PROGRAM POU_Lubrication
VAR
END_VAR

END_PROGRAM

(* stored: Version 1.1.0.1, ProductVersion 3.1.4024.12
   POU POU_Lubrication: Id {3a0089b1-665f-404c-aeec-fa8a66974b1b}, SpecialFunc None *)
